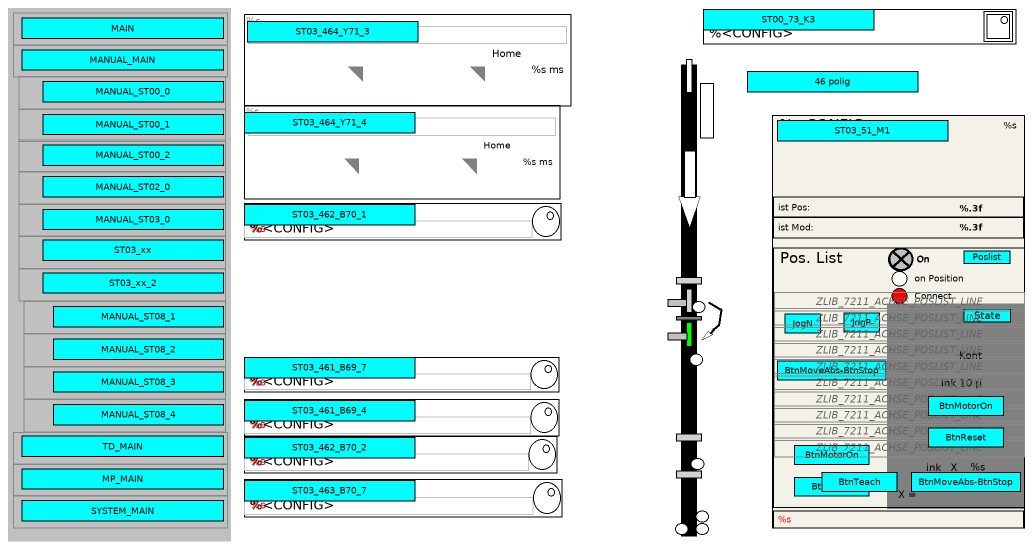
embedded screen at (3,115)-(226,648): M0000_Manual
embedded screen at (239,121)-(566,213): ZLIB_VALVE_1_SENSORS
embedded screen at (239,212)-(555,306): ZLIB_VALVE_1_SENSORS
embedded screen at (239,543)-(552,580): VDIGIN
embedded screen at (239,310)-(556,347): VDIGIN
embedded screen at (239,506)-(554,543): VDIGIN
embedded screen at (239,586)-(557,624): VDIGIN
embedded screen at (239,464)-(554,499): VDIGIN
embedded screen at (767,222)-(1021,635): ZLIB_7211_Achse
embedded screen at (646,161)-(716,643): ZUFUEHRUNG_46POL
rectangle at (742,178)-(913,199): text "46 polig"; invisible if TRUE
rectangle at (239,219)-(410,240): text "ST03_464_Y71_4"; invisible if TRUE
rectangle at (242,128)-(413,149): text "ST03_464_Y71_3"; invisible if TRUE
rectangle at (239,311)-(410,332): text "ST03_462_B70_1"; invisible if TRUE
rectangle at (239,507)-(410,528): text "ST03_461_B69_4"; invisible if TRUE
rectangle at (239,544)-(410,565): text "ST03_462_B70_2"; invisible if TRUE
rectangle at (239,587)-(410,608): text "ST03_463_B70_7"; invisible if TRUE
rectangle at (239,464)-(410,485): text "ST03_461_B69_7"; invisible if TRUE
rectangle at (772,227)-(943,248): text "ST03_51_M1"; invisible if TRUE
embedded screen at (698,116)-(1011,151): VDIGOUT_SMAL
rectangle at (698,116)-(869,137): text "ST00_73_K3"; invisible if TRUE
*)

(* Visualisation 01_ManualMode/ST03/MANUAL_ST03_9_2
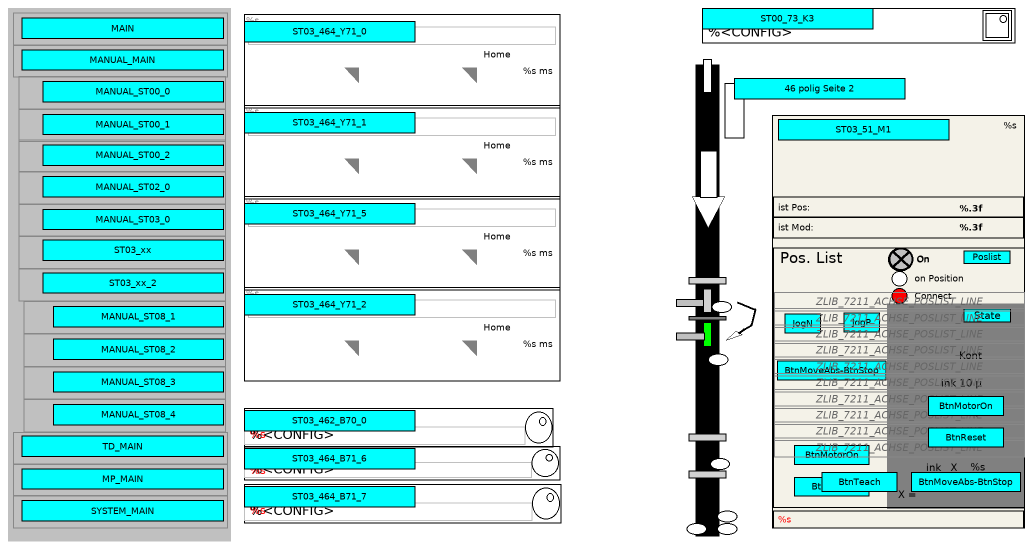
embedded screen at (3,115)-(226,648): M0000_Manual
embedded screen at (767,222)-(1021,635): ZLIB_7211_Achse
embedded screen at (646,161)-(750,643): ZUFUEHRUNG_46POL
rectangle at (729,185)-(900,206): text "46 polig Seite 2"; invisible if TRUE
embedded screen at (239,553)-(555,587): VDIGIN
embedded screen at (239,121)-(555,215): ZLIB_VALVE_1_SENSORS
rectangle at (239,128)-(410,149): text "ST03_464_Y71_0"; invisible if TRUE
rectangle at (239,555)-(410,576): text "ST03_464_B71_6"; invisible if TRUE
embedded screen at (239,212)-(555,306): ZLIB_VALVE_1_SENSORS
rectangle at (239,219)-(410,240): text "ST03_464_Y71_1"; invisible if TRUE
embedded screen at (239,394)-(555,488): ZLIB_VALVE_1_SENSORS
rectangle at (239,401)-(410,422): text "ST03_464_Y71_2"; invisible if TRUE
embedded screen at (239,303)-(555,397): ZLIB_VALVE_1_SENSORS
rectangle at (239,310)-(410,331): text "ST03_464_Y71_5"; invisible if TRUE
embedded screen at (239,515)-(548,554): VDIGIN
rectangle at (239,517)-(410,538): text "ST03_462_B70_0"; invisible if TRUE
rectangle at (773,226)-(944,247): text "ST03_51_M1"; invisible if TRUE
embedded screen at (239,591)-(556,630): VDIGIN
rectangle at (239,593)-(410,614): text "ST03_464_B71_7"; invisible if TRUE
embedded screen at (697,115)-(1010,150): VDIGOUT_SMAL
rectangle at (697,115)-(868,136): text "ST00_73_K3"; invisible if TRUE
*)

(* Visualisation 01_ManualMode/ST08/MANUAL_ST08_1
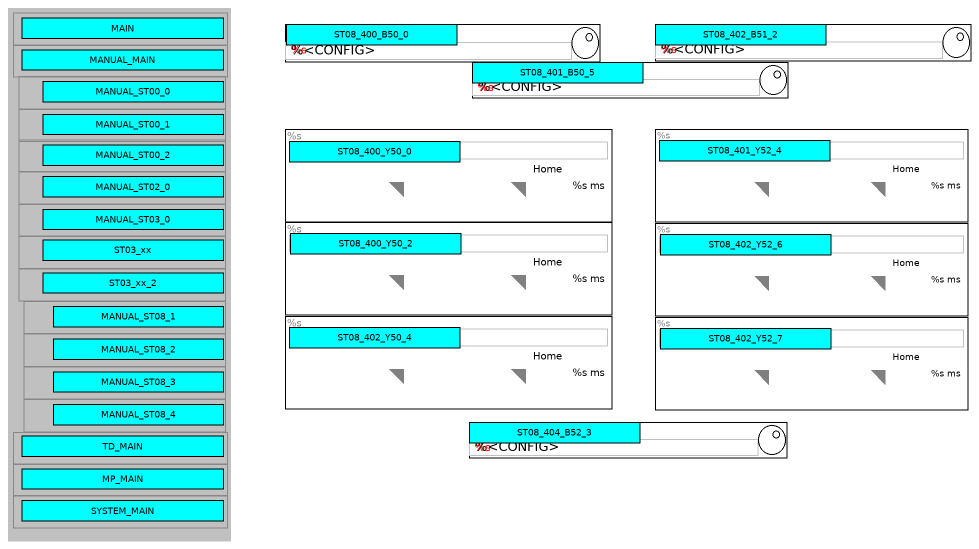
embedded screen at (3,115)-(226,648): M0000_Manual
embedded screen at (280,236)-(607,329): ZLIB_VALVE_1_SENSORS
embedded screen at (280,329)-(607,422): ZLIB_VALVE_1_SENSORS
embedded screen at (280,131)-(595,169): VDIGIN
embedded screen at (467,169)-(783,205): VDIGIN
embedded screen at (650,131)-(966,168): VDIGIN
embedded screen at (280,423)-(607,516): ZLIB_VALVE_1_SENSORS
embedded screen at (650,236)-(963,329): ZLIB_VALVE_1_SENSORS
embedded screen at (650,330)-(963,423): ZLIB_VALVE_1_SENSORS
embedded screen at (650,424)-(963,517): ZLIB_VALVE_1_SENSORS
embedded screen at (464,529)-(782,565): VDIGIN
rectangle at (281,131)-(452,152): text "ST08_400_B50_0"; invisible if TRUE
rectangle at (467,169)-(638,190): text "ST08_401_B50_5"; invisible if TRUE
rectangle at (650,131)-(821,152): text "ST08_402_B51_2"; invisible if TRUE
rectangle at (284,248)-(455,269): text "ST08_400_Y50_0"; invisible if TRUE
rectangle at (285,340)-(456,361): text "ST08_400_Y50_2"; invisible if TRUE
rectangle at (654,247)-(825,268): text "ST08_401_Y52_4"; invisible if TRUE
rectangle at (655,341)-(826,362): text "ST08_402_Y52_6"; invisible if TRUE
rectangle at (655,435)-(826,456): text "ST08_402_Y52_7"; invisible if TRUE
rectangle at (284,434)-(455,455): text "ST08_402_Y50_4"; invisible if TRUE
rectangle at (464,529)-(635,550): text "ST08_404_B52_3"; invisible if TRUE
*)

(* Visualisation 01_ManualMode/ST08/MANUAL_ST08_2
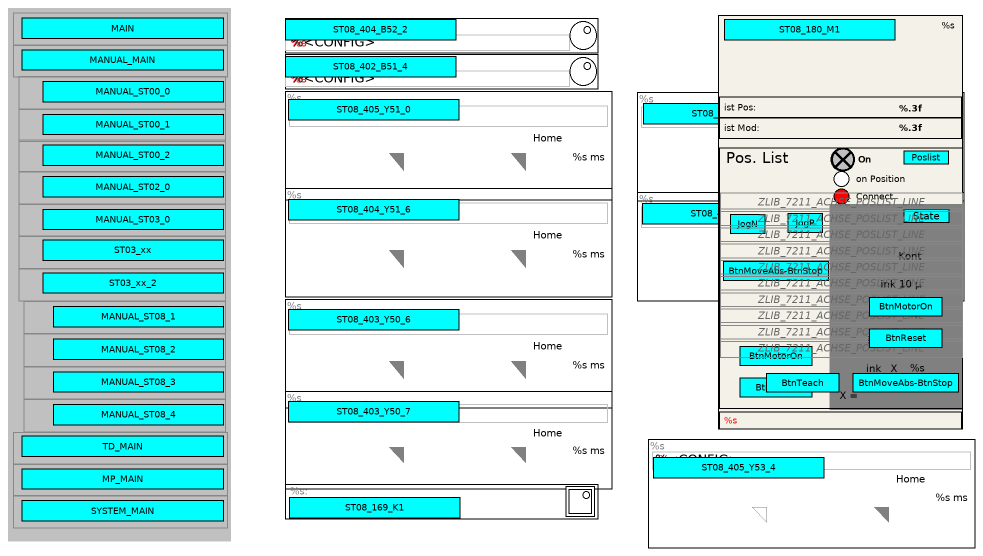
embedded screen at (3,115)-(226,648): M0000_Manual
embedded screen at (280,125)-(593,160): VDIGIN
embedded screen at (280,198)-(607,307): ZLIB_VALVE_1_SENSORS
embedded screen at (280,295)-(607,404): ZLIB_VALVE_1_SENSORS
embedded screen at (643,546)-(970,655): ZLIB_VALVE_2_SENSORS
embedded screen at (280,406)-(607,515): ZLIB_VALVE_1_SENSORS
embedded screen at (280,498)-(607,596): ZLIB_VALVE_1_SENSORS
embedded screen at (280,161)-(593,196): VDIGIN
embedded screen at (632,199)-(959,308): ZLIB_VALVE_1_SENSORS
rectangle at (638,210)-(809,231): text "ST08_404_Y53_0"; invisible if TRUE
embedded screen at (632,299)-(959,408): ZLIB_VALVE_1_SENSORS
rectangle at (637,310)-(808,331): text "ST08_404_Y53_2"; invisible if TRUE
embedded screen at (713,122)-(959,536): ZLIB_7211_Achse
embedded screen at (280,591)-(593,626): VDIGOUT_SMAL
rectangle at (280,126)-(451,147): text "ST08_404_B52_2"; invisible if TRUE
rectangle at (280,163)-(451,184): text "ST08_402_B51_4"; invisible if TRUE
rectangle at (283,206)-(454,227): text "ST08_405_Y51_0"; invisible if TRUE
rectangle at (283,306)-(454,327): text "ST08_404_Y51_6"; invisible if TRUE
rectangle at (283,416)-(454,437): text "ST08_403_Y50_6"; invisible if TRUE
rectangle at (283,508)-(454,529): text "ST08_403_Y50_7"; invisible if TRUE
rectangle at (284,604)-(455,625): text "ST08_169_K1"; invisible if TRUE
rectangle at (648,564)-(819,585): text "ST08_405_Y53_4"; invisible if TRUE
rectangle at (719,126)-(890,147): text "ST08_180_M1"; invisible if TRUE
*)

(* Visualisation 01_ManualMode/ST08/MANUAL_ST08_3
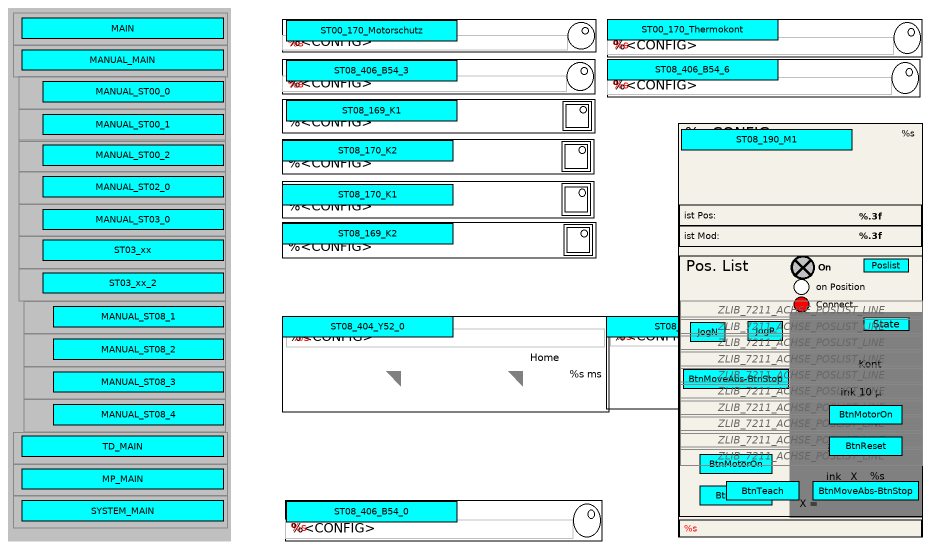
embedded screen at (3,115)-(226,648): M0000_Manual
embedded screen at (277,206)-(590,240): VDIGOUT_SMAL
embedded screen at (277,329)-(591,365): VDIGOUT_SMAL
embedded screen at (277,288)-(589,325): VDIGOUT_SMAL
embedded screen at (277,246)-(589,281): VDIGOUT_SMAL
embedded screen at (602,126)-(917,164): VDIGIN
embedded screen at (277,126)-(591,159): VDIGIN
embedded screen at (280,607)-(597,648): VDIGIN
embedded screen at (277,166)-(590,201): VDIGIN
embedded screen at (601,423)-(914,516): ZLIB_VALVE_1_SENSORS
embedded screen at (277,423)-(604,519): ZLIB_VALVE_1_SENSORS
rectangle at (601,423)-(772,444): text "ST08_406_Y52_3"; invisible if TRUE
rectangle at (277,423)-(448,444): text "ST08_404_Y52_0"; invisible if TRUE
rectangle at (281,207)-(452,228): text "ST08_169_K1"; invisible if TRUE
rectangle at (277,330)-(448,351): text "ST08_169_K2"; invisible if TRUE
rectangle at (277,291)-(448,312): text "ST08_170_K1"; invisible if TRUE
rectangle at (277,247)-(448,268): text "ST08_170_K2"; invisible if TRUE
rectangle at (281,127)-(452,148): text "ST00_170_Motorschutz"; invisible if TRUE
rectangle at (602,126)-(773,147): text "ST00_170_Thermokont"; invisible if TRUE
rectangle at (281,608)-(452,629): text "ST08_406_B54_0"; invisible if TRUE
rectangle at (281,167)-(452,188): text "ST08_406_B54_3"; invisible if TRUE
embedded screen at (602,166)-(915,204): VDIGIN
rectangle at (602,166)-(773,187): text "ST08_406_B54_6"; invisible if TRUE
embedded screen at (673,230)-(919,644): ZLIB_7211_Achse
rectangle at (676,236)-(847,257): text "ST08_190_M1"; invisible if TRUE
*)

(* Visualisation 01_ManualMode/ST08/MANUAL_ST08_4
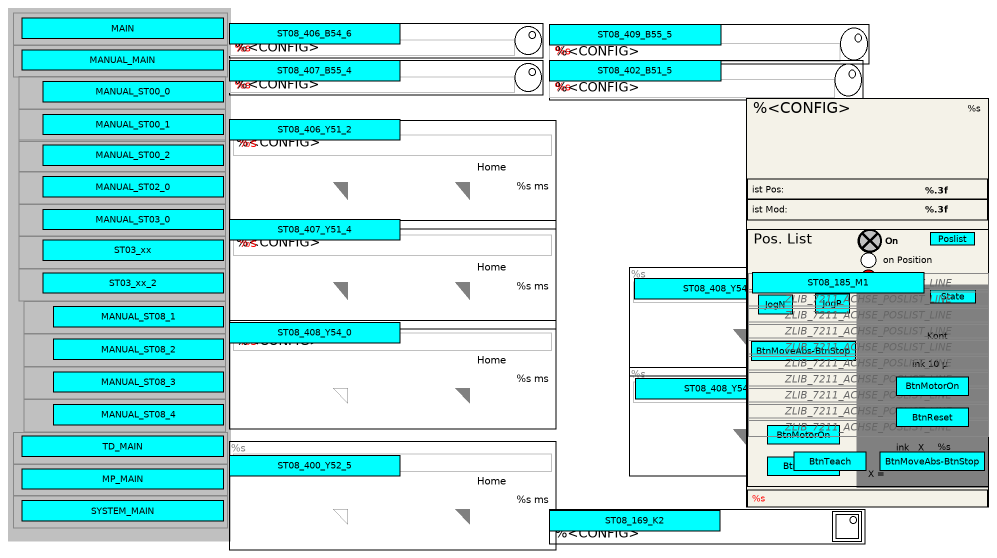
embedded screen at (3,115)-(226,648): M0000_Manual
embedded screen at (224,427)-(551,536): ZLIB_VALVE_2_SENSORS
embedded screen at (224,130)-(538,165): VDIGIN
embedded screen at (224,227)-(551,336): ZLIB_VALVE_1_SENSORS
embedded screen at (224,327)-(551,436): ZLIB_VALVE_1_SENSORS
embedded screen at (544,131)-(864,171): VDIGIN
embedded screen at (224,548)-(551,657): ZLIB_VALVE_2_SENSORS
embedded screen at (544,167)-(858,207): VDIGIN
embedded screen at (624,374)-(951,483): ZLIB_VALVE_1_SENSORS
rectangle at (629,385)-(801,406): text "ST08_408_Y54_2"; invisible if TRUE
embedded screen at (624,474)-(951,583): ZLIB_VALVE_1_SENSORS
rectangle at (630,485)-(802,506): text "ST08_408_Y54_4"; invisible if TRUE
embedded screen at (741,205)-(985,614): ZLIB_7211_Achse
embedded screen at (224,167)-(538,202): VDIGIN
embedded screen at (544,616)-(860,651): VDIGOUT_SMAL
rectangle at (224,562)-(395,583): text "ST08_400_Y52_5"; invisible if TRUE
rectangle at (544,617)-(715,638): text "ST08_169_K2"; invisible if TRUE
rectangle at (224,429)-(395,450): text "ST08_408_Y54_0"; invisible if TRUE
rectangle at (224,326)-(395,347): text "ST08_407_Y51_4"; invisible if TRUE
rectangle at (224,226)-(395,247): text "ST08_406_Y51_2"; invisible if TRUE
rectangle at (224,130)-(395,151): text "ST08_406_B54_6"; invisible if TRUE
rectangle at (224,167)-(395,188): text "ST08_407_B55_4"; invisible if TRUE
rectangle at (544,131)-(716,152): text "ST08_409_B55_5"; invisible if TRUE
rectangle at (544,167)-(716,188): text "ST08_402_B51_5"; invisible if TRUE
rectangle at (747,379)-(919,400): text "ST08_185_M1"; invisible if TRUE
*)

(* Visualisation 00_Main/MASTER_MAIN
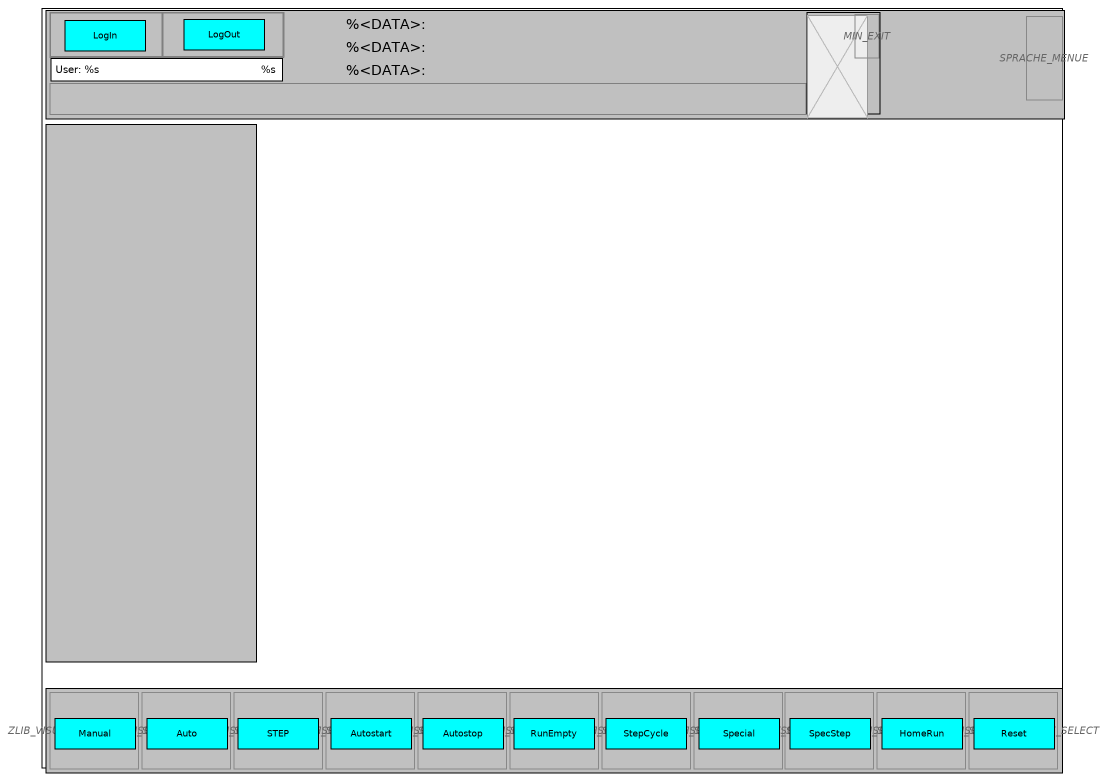
embedded screen at (8,684)-(97,761): ZLIB_VISUBUTTON_MODE_SELECT
embedded screen at (100,684)-(189,761): ZLIB_VISUBUTTON_MODE_SELECT
embedded screen at (192,684)-(281,761): ZLIB_VISUBUTTON_MODE_SELECT
embedded screen at (284,684)-(373,761): ZLIB_VISUBUTTON_MODE_SELECT
embedded screen at (376,684)-(465,761): ZLIB_VISUBUTTON_MODE_SELECT
embedded screen at (468,684)-(557,761): ZLIB_VISUBUTTON_MODE_SELECT
embedded screen at (560,684)-(649,761): ZLIB_VISUBUTTON_MODE_SELECT
embedded screen at (652,684)-(741,761): ZLIB_VISUBUTTON_MODE_SELECT
embedded screen at (835,684)-(924,761): ZLIB_VISUBUTTON_MODE_SELECT
embedded screen at (927,684)-(1016,761): ZLIB_VISUBUTTON_MODE_SELECT
rectangle at (247,29)-(386,49): text "%<DATA>:"; shows 'ArtNo'
rectangle at (247,6)-(386,26): text "%<DATA>:"; shows 'TypeName'
rectangle at (247,52)-(386,72): text "%<DATA>:"; shows 'TypeDescription'
rectangle at (9,50)-(241,73): text "User: %s"; shows UserLoginHandler.CurrentUser.UserName
embedded screen at (8,4)-(121,49): ZLIB_VISUBUTTON_S18
embedded screen at (120,4)-(242,49): ZLIB_VISUBUTTON_S18
embedded screen at (8,75)-(764,106): ZLIB_ShowMessageButton
embedded screen at (743,684)-(832,761): ZLIB_VISUBUTTON_MODE_SELECT
rectangle at (13,710)-(94,741): text "Manual"; invisible if TRUE
rectangle at (105,710)-(186,741): text "Auto"; invisible if TRUE
rectangle at (196,710)-(277,741): text "STEP"; invisible if TRUE
rectangle at (289,710)-(370,741): text "Autostart"; invisible if TRUE
rectangle at (381,710)-(462,741): text "Autostop"; invisible if TRUE
rectangle at (472,710)-(553,741): text "RunEmpty"; invisible if TRUE
rectangle at (564,710)-(645,741): text "StepCycle"; invisible if TRUE
rectangle at (657,710)-(738,741): text "Special"; invisible if TRUE
rectangle at (748,710)-(829,741): text "SpecStep"; invisible if TRUE
rectangle at (840,710)-(921,741): text "HomeRun"; invisible if TRUE
rectangle at (932,710)-(1013,741): text "Reset"; invisible if TRUE
rectangle at (142,11)-(223,42): text "LogOut"; invisible if TRUE
rectangle at (23,12)-(104,43): text "LogIn"; invisible if TRUE
rectangle at (157,52)-(239,71): text "%s"; shows UserLoginHandler.s_AutoLoggedOut
group at (765,4)-(1021,110)
  bitmap at (3,3)-(213,106): c:\twincat\plc\VisuBmp\ept_logo.jpg
  embedded screen at (168,2)-(253,46): MIN_EXIT
  embedded screen at (765,4)-(891,88): SPRACHE_MENUE
5 more shapes without text or variables
6 elements of other kinds (tables, trends, ...) not read
*)

(* Visualisation zLibrary/ept/MIN_EXIT
2 elements of other kinds (tables, trends, ...) not read
*)

(* Visualisation 03_MachPara/MP_DATE
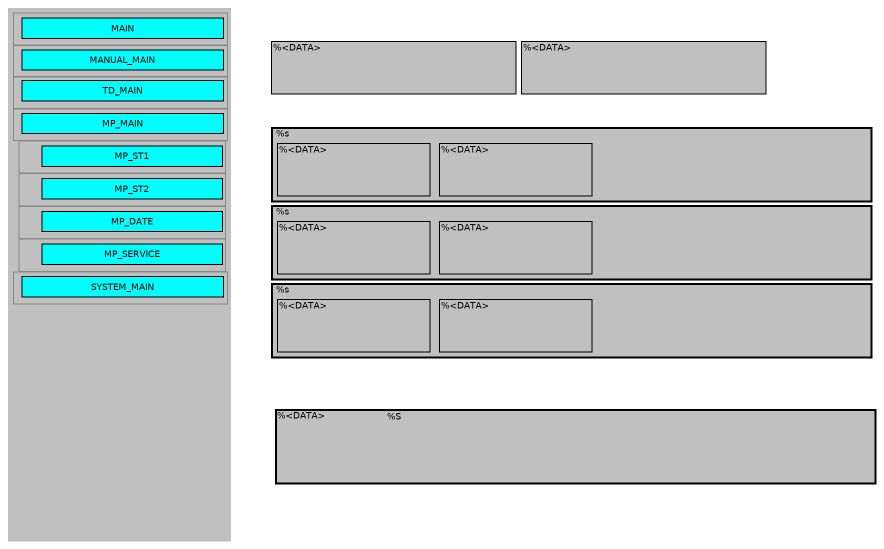
rectangle at (266,390)-(867,465): text "%s"; shows .MP.ShiftData.Shift[3].ShiftName; alarm colour if .MP.ShiftData.Shift[3].ShiftActive
rectangle at (266,312)-(867,387): text "%s"; shows .MP.ShiftData.Shift[2].ShiftName; alarm colour if .MP.ShiftData.Shift[2].ShiftActive
rectangle at (266,234)-(867,309): text "%s"; shows .MP.ShiftData.Shift[1].ShiftName; alarm colour if .MP.ShiftData.Shift[1].ShiftActive
rectangle at (516,148)-(761,201): text "%<DATA>"; shows 'Uhrzeit'
rectangle at (266,148)-(511,201): text "%<DATA>"; shows 'Datum'
embedded screen at (3,115)-(226,648): M0002_Machpara
rectangle at (272,250)-(425,303): text "%<DATA>"; shows 'Uhrzeit Start'
rectangle at (434,250)-(587,303): text "%<DATA>"; shows 'Uhrzeit Ende'
rectangle at (272,328)-(425,381): text "%<DATA>"; shows 'Uhrzeit Start'
rectangle at (434,328)-(587,381): text "%<DATA>"; shows 'Uhrzeit Ende'
rectangle at (272,406)-(425,459): text "%<DATA>"; shows 'Uhrzeit Start'
rectangle at (434,406)-(587,459): text "%<DATA>"; shows 'Uhrzeit Ende'
rectangle at (270,516)-(871,591): text "%<DATA>"; shows 'Aktuelle Schicht'; alarm colour if .MP.ShiftData.Activeshift.ShiftActive
rectangle at (380,515)-(511,532): text "%S"; shows .MP.ShiftData.Activeshift.ShiftName
35 elements of other kinds (tables, trends, ...) not read
*)

(* Visualisation 03_MachPara/MP_SERVICE
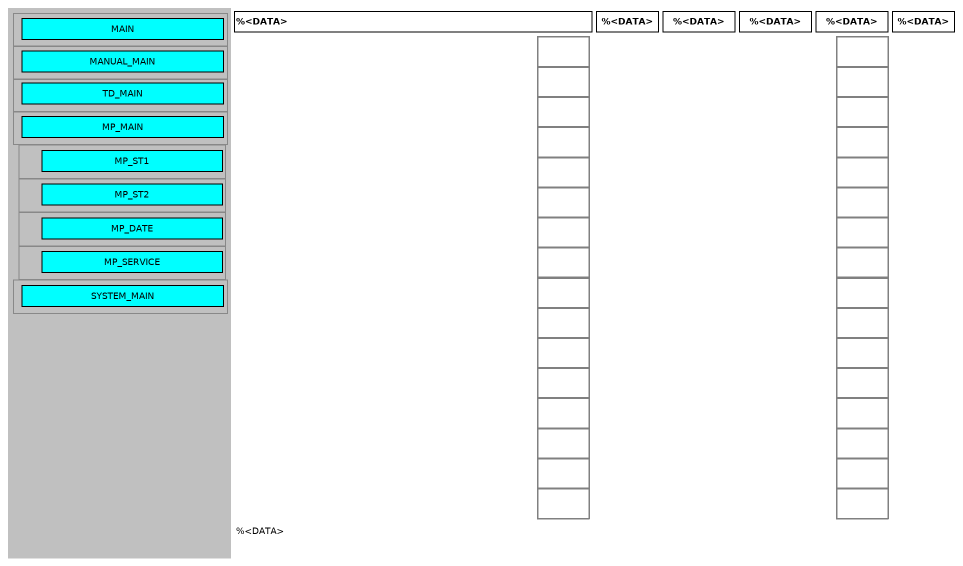
embedded screen at (3,115)-(226,665): M0002_Machpara
embedded screen at (229,118)-(1011,651): ZLIB_SERVICELIST
*)

(* Visualisation 03_MachPara/MP_ST1
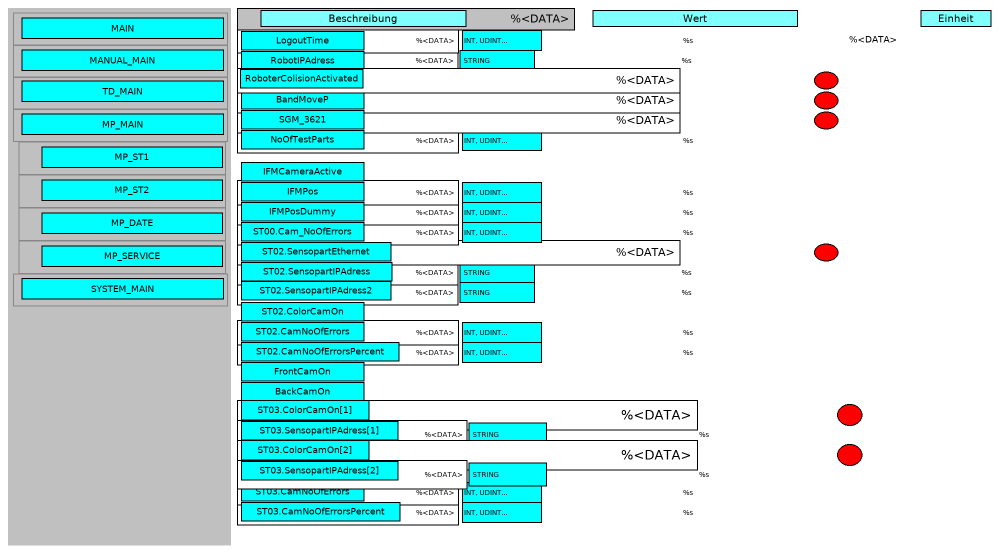
embedded screen at (3,115)-(226,652): M0002_Machpara
rectangle at (842,136)-(960,157): text "%<DATA>"; shows '0_deaktiv'
embedded screen at (232,607)-(833,632): Data_DEZIMAL
embedded screen at (232,587)-(833,612): Data_DEZIMAL
embedded screen at (232,447)-(833,472): Data_DEZIMAL
embedded screen at (232,427)-(833,452): Data_DEZIMAL
embedded screen at (232,387)-(833,412): Data_STRING
embedded screen at (232,367)-(833,392): Data_STRING
embedded screen at (232,347)-(833,372): Data_BOOL
embedded screen at (232,327)-(833,352): Data_DEZIMAL
embedded screen at (232,307)-(833,332): Data_DEZIMAL
embedded screen at (232,287)-(833,312): Data_DEZIMAL
embedded screen at (232,235)-(833,260): Data_DEZIMAL
embedded screen at (232,215)-(833,240): Data_BOOL
embedded screen at (232,195)-(833,220): Data_BOOL
embedded screen at (232,155)-(833,180): Data_STRING
embedded screen at (232,135)-(833,160): Data_DEZIMAL
rectangle at (236,158)-(359,177): text "RobotIPAdress"; invisible if TRUE
rectangle at (236,197)-(359,216): text "BandMoveP"; invisible if TRUE
rectangle at (236,217)-(359,236): text "SGM_3621"; invisible if TRUE
rectangle at (236,369)-(387,388): text "ST02.SensopartIPAdress"; invisible if TRUE
rectangle at (236,349)-(386,368): text "ST02.SensopartEthernet"; invisible if TRUE
rectangle at (236,269)-(359,288): text "IFMCameraActive"; invisible if TRUE
rectangle at (236,309)-(359,328): text "IFMPosDummy"; invisible if TRUE
rectangle at (236,388)-(386,407): text "ST02.SensopartIPAdress2"; invisible if TRUE
rectangle at (236,449)-(394,468): text "ST02.CamNoOfErrorsPercent"; invisible if TRUE
rectangle at (236,469)-(359,488): text "FrontCamOn"; invisible if TRUE
rectangle at (236,609)-(395,628): text "ST03.CamNoOfErrorsPercent"; invisible if TRUE
rectangle at (236,237)-(359,256): text "NoOfTestParts"; invisible if TRUE
rectangle at (236,329)-(359,348): text "ST00.Cam_NoOfErrors"; invisible if TRUE
rectangle at (236,429)-(359,448): text "ST02.CamNoOfErrors"; invisible if TRUE
rectangle at (236,489)-(359,508): text "BackCamOn"; shows 'BackCamOn'; invisible if TRUE
rectangle at (236,589)-(359,608): text "ST03.CamNoOfErrors"; invisible if TRUE
rectangle at (236,289)-(359,308): text "IFMPos"; invisible if TRUE
rectangle at (236,138)-(359,157): text "LogoutTime"; invisible if TRUE
rectangle at (236,409)-(359,428): text "ST02.ColorCamOn"; invisible if TRUE
embedded screen at (232,175)-(833,200): Data_BOOL
rectangle at (235,176)-(358,195): text "RoboterColisionActivated"; shows 'BackCamOn'; invisible if TRUE
embedded screen at (232,115)-(986,137): DATA_HEADER_BEER
embedded screen at (232,507)-(857,537): Data_BOOL
embedded screen at (232,527)-(857,556): Data_STRING
rectangle at (236,528)-(393,547): text "ST03.SensopartIPAdress[1]"; invisible if TRUE
rectangle at (236,507)-(364,527): text "ST03.ColorCamOn[1]"; invisible if TRUE
embedded screen at (232,547)-(857,577): Data_BOOL
embedded screen at (232,567)-(857,596): Data_STRING
rectangle at (236,568)-(393,587): text "ST03.SensopartIPAdress[2]"; invisible if TRUE
rectangle at (236,547)-(364,567): text "ST03.ColorCamOn[2]"; invisible if TRUE
4 elements of other kinds (tables, trends, ...) not read
*)

(* Visualisation 03_MachPara/MP_ST2
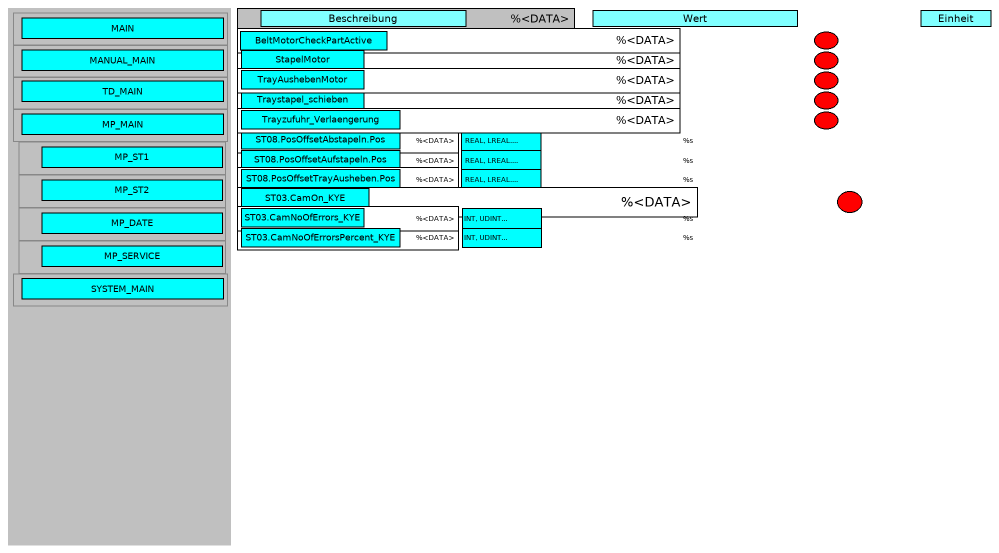
embedded screen at (3,115)-(226,652): M0002_Machpara
embedded screen at (232,115)-(986,137): DATA_HEADER_BEER
embedded screen at (232,255)-(833,280): Data_DEZIMAL_REAL
embedded screen at (232,235)-(833,260): Data_DEZIMAL_REAL
embedded screen at (232,195)-(833,220): Data_BOOL
embedded screen at (232,155)-(833,180): Data_BOOL
embedded screen at (232,135)-(833,160): Data_BOOL
rectangle at (236,197)-(359,216): text "Traystapel_schieben"; invisible if TRUE
rectangle at (236,157)-(359,176): text "StapelMotor"; invisible if TRUE
rectangle at (236,237)-(395,256): text "ST08.PosOffsetAbstapeln.Pos"; invisible if TRUE
rectangle at (236,257)-(395,276): text "ST08.PosOffsetAufstapeln.Pos"; invisible if TRUE
rectangle at (235,138)-(382,157): text "BeltMotorCheckPartActive"; invisible if TRUE
embedded screen at (232,175)-(833,200): Data_BOOL
rectangle at (236,177)-(359,196): text "TrayAushebenMotor"; invisible if TRUE
embedded screen at (232,274)-(833,299): Data_DEZIMAL_REAL
rectangle at (236,276)-(395,295): text "ST08.PosOffsetTrayAusheben.Pos"; invisible if TRUE
embedded screen at (232,215)-(833,240): Data_BOOL
rectangle at (236,217)-(395,236): text "Trayzufuhr_Verlaengerung"; invisible if TRUE
embedded screen at (232,294)-(857,324): Data_BOOL
rectangle at (236,295)-(364,315): text "ST03.CamOn_KYE"; invisible if TRUE
embedded screen at (232,332)-(833,357): Data_DEZIMAL
embedded screen at (232,313)-(833,338): Data_DEZIMAL
rectangle at (236,335)-(395,354): text "ST03.CamNoOfErrorsPercent_KYE"; invisible if TRUE
rectangle at (236,315)-(359,334): text "ST03.CamNoOfErrors_KYE"; invisible if TRUE
*)

(* Visualisation zLibrary/X_MachSpec/PARTRESULT
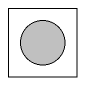
ellipse at (12,12)-(57,57): invisible if ($PartResult$ MOD 10) = 0; alarm colour if ($PartResult$ MOD 10) <> 1
ellipse at (12,12)-(57,57): invisible if ($PartResult$ MOD 10) <> 4
ellipse at (12,12)-(57,57): invisible if ($PartResult$ MOD 10) <> 5
ellipse at (12,12)-(57,57): invisible if ($PartResult$ MOD 10) <> 0
1 more shapes without text or variables
*)

(* Visualisation zLibrary/ept/Pruefteile/PRUEFTEILEN_CZ
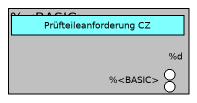
rectangle at (0,0)-(181,86): text "%<BASIC>"; shows 'auto_Prüfteileanforderung'
rectangle at (156,37)-(179,59): text "%d"; shows ST03_Main.CTR; invisible if gTakeTestParts=FALSE AND gTakeTestPartsAuto=FALSE; alarm colour if gTakeTestParts OR gTakeTestPartsAuto
rectangle at (18,61)-(153,82): text "%<BASIC>"; shows 'Rutsche belegt'; invisible if .TD.TestpartBilister
ellipse at (156,61)-(167,72): invisible if .TD.TestpartBilister; alarm colour if ST03_8_75_B13_5.BitInToCheck
ellipse at (156,73)-(167,84): invisible if .TD.TestpartBilister; alarm colour if ST03_8_75_B13_6.BitInToCheck
rectangle at (3,7)-(176,27): text "Prüfteileanforderung CZ"; invisible if TRUE
1 elements of other kinds (tables, trends, ...) not read
*)

(* Visualisation zLibrary/ept/Pruefteile/PRUEFTEILEN_DE
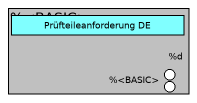
rectangle at (0,0)-(181,86): text "%<BASIC>"; shows 'Prüfteileanforderung'
rectangle at (156,37)-(179,59): text "%d"; shows ST03_Main.CTR; invisible if gTakeTestParts=FALSE AND gTakeTestPartsAuto=FALSE; alarm colour if gTakeTestParts OR gTakeTestPartsAuto
rectangle at (19,61)-(153,82): text "%<BASIC>"; shows 'Rutsche belegt'; invisible if .TD.TestpartBilister
ellipse at (156,61)-(167,72): invisible if .TD.TestpartBilister; alarm colour if ST03_8_75_B13_5.BitInToCheck
ellipse at (156,73)-(167,84): invisible if .TD.TestpartBilister; alarm colour if ST03_8_75_B13_6.BitInToCheck
rectangle at (3,7)-(176,27): text "Prüfteileanforderung DE"; invisible if TRUE
1 elements of other kinds (tables, trends, ...) not read
*)

(* Visualisation zLibrary/ept/Pruefteile/PRUEFTEILENTNAHME
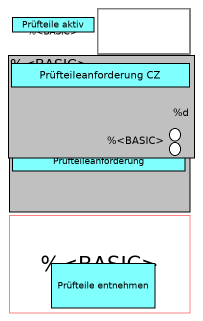
embedded screen at (89,5)-(182,51): ZLIB_VISUBUTTON_S24
rectangle at (1,8)-(88,49): text "%<BASIC>"; shows 'Prüfteile aktiv'; invisible if NOT gTakeTestParts AND NOT gTakeTestPartsAuto; alarm colour if gTakeTestParts OR gTakeTestPartsAuto
rectangle at (1,212)-(182,310): text "%<BASIC>"; shows 'Prüfteile entnehmen'; invisible if NOT ST03_Main.TestPartsRemove; taps gTakeTestPartsFinished
rectangle at (43,260)-(147,305): text "Prüfteile entnehmen"; invisible if TRUE
rectangle at (4,14)-(86,29): text "Prüfteile aktiv"; invisible if TRUE
rectangle at (1,141)-(182,209): text "%<BASIC>"; shows 'Teile seit letzten Test'
rectangle at (4,148)-(177,168): text "Prüfteileanforderung"; invisible if TRUE
embedded screen at (0,52)-(187,155): PRUEFTEILEN_CZ
2 elements of other kinds (tables, trends, ...) not read
*)

(* Visualisation zLibrary/X_MachSpec/RoundTable/ROUNDTABLE
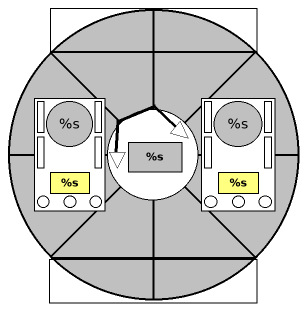
polyline at (147,3)-(147,291): invisible if (ST02_DT_62_B81.ValveSensor OR ST02_DT_62_B91.ValveSensor)
polyline at (2,147)-(292,147): invisible if (ST02_DT_62_B81.ValveSensor OR ST02_DT_62_B91.ValveSensor)
polyline at (44,44)-(249,249): invisible if NOT (ST02_DT_62_B81.ValveSensor OR ST02_DT_62_B91.ValveSensor)
polyline at (44,44)-(249,249): invisible if NOT (ST02_DT_62_B81.ValveSensor OR ST02_DT_62_B91.ValveSensor)
embedded screen at (195,90)-(269,203): RoundTableNest
embedded screen at (28,90)-(99,203): ROUNDTABLENEST
polygon at (103,144)-(119,160): alarm colour if ST02_62_Y6.MoveWork
rounded rectangle at (122,134)-(176,164): text "%s"; shows MachineStates.CycleTimeHelp
polygon at (164,113)-(182,130): alarm colour if ST02_62_Y6.MoveInit
7 more shapes without text or variables
*)

(* Visualisation zLibrary/X_MachSpec/RoundTable/ROUNDTABLE_1
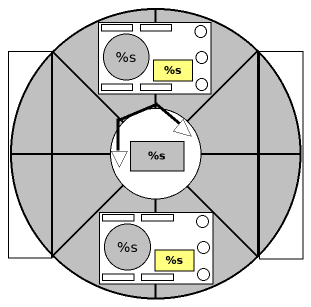
polyline at (147,3)-(147,291): invisible if (ST02_DT_62_B81.ValveSensor OR ST02_DT_62_B91.ValveSensor)
polyline at (2,147)-(292,147): invisible if (ST02_DT_62_B81.ValveSensor OR ST02_DT_62_B91.ValveSensor)
polyline at (44,44)-(249,249): invisible if NOT (ST02_DT_62_B81.ValveSensor OR ST02_DT_62_B91.ValveSensor)
polyline at (44,44)-(249,249): invisible if NOT (ST02_DT_62_B81.ValveSensor OR ST02_DT_62_B91.ValveSensor)
embedded screen at (90,14)-(203,87): RoundTableNest_1
embedded screen at (91,204)-(205,277): ROUNDTABLENEST_1
polygon at (103,144)-(119,160): alarm colour if ST02_62_Y6.MoveWork
rounded rectangle at (122,134)-(176,164): text "%s"; shows MachineStates.CycleTimeHelp
polygon at (165,112)-(183,129): alarm colour if ST02_62_Y6.MoveInit
7 more shapes without text or variables
*)

(* Visualisation zLibrary/X_MachSpec/RoundTable/ROUNDTABLENEST
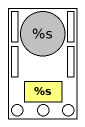
ellipse at (12,3)-(57,48): text "%s"; shows $NestNo$; invisible if NOT MP.ST02.TableData[$NestNo$].ProcessData.Part; alarm colour if MP.ST02.TableData[$NestNo$].ProcessData.Result >11; toggles MP.ST02.TableData[$NestNo$].ProcessData.Part
ellipse at (12,3)-(57,48): text "%s"; shows $NestNo$; invisible if MP.ST02.TableData[$NestNo$].ProcessData.Part; toggles MP.ST02.TableData[$NestNo$].ProcessData.Part
rectangle at (16,73)-(54,94): text "%s"; shows MP.ST02.TableData[$NestNo$].ProcessData.Result; editable
rectangle at (3,38)-(10,69): invisible if NOT MP.ST02.TableData[$NestNo$].ProcessData.Part OR MP.ST02.TableData[$NestNo$].ProcessData.Result >=19; alarm colour if MP.ST02.TableData[$NestNo$].ProcessData.Result >=1
rectangle at (3,3)-(10,34): invisible if NOT MP.ST02.TableData[$NestNo$].ProcessData.Part OR MP.ST02.TableData[$NestNo$].ProcessData.Result >=19; alarm colour if MP.ST02.TableData[$NestNo$].ProcessData.Result >=1
rectangle at (59,38)-(66,69): invisible if NOT MP.ST02.TableData[$NestNo$].ProcessData.Part OR MP.ST02.TableData[$NestNo$].ProcessData.Result >=19; alarm colour if MP.ST02.TableData[$NestNo$].ProcessData.Result >=11
rectangle at (59,3)-(66,34): invisible if NOT MP.ST02.TableData[$NestNo$].ProcessData.Part OR MP.ST02.TableData[$NestNo$].ProcessData.Result >=19; alarm colour if MP.ST02.TableData[$NestNo$].ProcessData.Result >=11
ellipse at (3,96)-(15,108): invisible if MP.ST02.TableData[$NestNo$].ProcessData.Nest_Nr = 0; alarm colour if ST02_Schwenkarm[MP.ST02.TableData[$NestNo$].ProcessData.Nest_Nr].ST02_90_0_sens
ellipse at (29,96)-(41,108): invisible if MP.ST02.TableData[$NestNo$].ProcessData.Nest_Nr = 0; alarm colour if ST02_Schwenkarm[MP.ST02.TableData[$NestNo$].ProcessData.Nest_Nr].ST02_90_sens
ellipse at (54,96)-(66,108): invisible if MP.ST02.TableData[$NestNo$].ProcessData.Nest_Nr = 0; alarm colour if ST02_Schwenkarm[MP.ST02.TableData[$NestNo$].ProcessData.Nest_Nr].ST02_90_180_sens
1 more shapes without text or variables
1 elements of other kinds (tables, trends, ...) not read
*)

(* Visualisation zLibrary/X_MachSpec/RoundTable/ROUNDTABLENEST_1
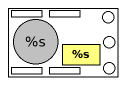
ellipse at (5,12)-(50,57): text "%s"; shows $NestNo$; invisible if NOT MP.ST02.TableData[$NestNo$].ProcessData.Part; alarm colour if MP.ST02.TableData[$NestNo$].ProcessData.Result >=99; toggles MP.ST02.TableData[$NestNo$].ProcessData.Part
ellipse at (5,12)-(50,57): text "%s"; shows $NestNo$; invisible if MP.ST02.TableData[$NestNo$].ProcessData.Part; toggles MP.ST02.TableData[$NestNo$].ProcessData.Part
rectangle at (54,37)-(92,58): text "%s"; shows MP.ST02.TableData[$NestNo$].ProcessData.Result; editable
rectangle at (41,60)-(72,67): invisible if NOT MP.ST02.TableData[$NestNo$].ProcessData.Part OR MP.ST02.TableData[$NestNo$].ProcessData.Result >=19; alarm colour if MP.ST02.TableData[$NestNo$].ProcessData.Result >=1
rectangle at (3,60)-(34,67): invisible if NOT MP.ST02.TableData[$NestNo$].ProcessData.Part OR MP.ST02.TableData[$NestNo$].ProcessData.Result >=19; alarm colour if MP.ST02.TableData[$NestNo$].ProcessData.Result >=1
rectangle at (41,3)-(72,10): invisible if NOT MP.ST02.TableData[$NestNo$].ProcessData.Part OR MP.ST02.TableData[$NestNo$].ProcessData.Result >=19; alarm colour if MP.ST02.TableData[$NestNo$].ProcessData.Result >=11
rectangle at (3,3)-(34,10): invisible if NOT MP.ST02.TableData[$NestNo$].ProcessData.Part OR MP.ST02.TableData[$NestNo$].ProcessData.Result >=19; alarm colour if MP.ST02.TableData[$NestNo$].ProcessData.Result >=11
ellipse at (95,55)-(107,67): invisible if MP.ST02.TableData[$NestNo$].ProcessData.Nest_Nr = 0; alarm colour if ST02_Schwenkarm[MP.ST02.TableData[$NestNo$].ProcessData.Nest_Nr].ST02_90_0_sens
ellipse at (95,29)-(107,41): invisible if MP.ST02.TableData[$NestNo$].ProcessData.Nest_Nr = 0; alarm colour if ST02_Schwenkarm[MP.ST02.TableData[$NestNo$].ProcessData.Nest_Nr].ST02_90_sens
ellipse at (94,4)-(106,16): invisible if MP.ST02.TableData[$NestNo$].ProcessData.Nest_Nr = 0; alarm colour if ST02_Schwenkarm[MP.ST02.TableData[$NestNo$].ProcessData.Nest_Nr].ST02_90_180_sens
1 more shapes without text or variables
1 elements of other kinds (tables, trends, ...) not read
*)

(* Visualisation zLibrary/X_MachSpec/RoundTable/ROUNDTABLENESTNR
ellipse at (0,0)-(45,45): text "%s"; shows MP.ST02.TableData[$NestNo$].ProcessData.Nest_Nr; alarm colour if MP.ST02.DeactivatedNests[MP.ST02.TableData[$NestNo$].ProcessData.Nest_Nr]
*)

(* Visualisation zLibrary/X_MachSpec/Signs/SIGNS_ARROWDOWN
polygon at (0,72)-(48,120): alarm colour if $OnBit$
rectangle at (12,0)-(37,73): alarm colour if $OnBit$
*)

(* Visualisation zLibrary/X_MachSpec/Signs/SIGNS_ARROWLEFT
polygon at (0,0)-(48,48): alarm colour if $OnBit$
rectangle at (48,12)-(121,37): alarm colour if $OnBit$
*)

(* Visualisation zLibrary/X_MachSpec/Signs/SIGNS_ARROWRIGHT
polygon at (72,0)-(120,48): alarm colour if $OnBit$
rectangle at (0,12)-(73,37): alarm colour if $OnBit$
*)

(* Visualisation zLibrary/X_MachSpec/Signs/SIGNS_ARROWUP
polygon at (0,0)-(48,48): alarm colour if $OnBit$
rectangle at (12,48)-(37,121): alarm colour if $OnBit$
*)

(* Visualisation zLibrary/ept/Axis/SIGNS_AXIS
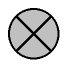
ellipse at (0,0)-(51,51): alarm colour if $Object$.on
polyline at (8,8)-(43,43): angle $Object$.sPos.lr_Mod /4
polyline at (8,8)-(43,43): angle $Object$.sPos.lr_Mod /4
*)

(* Visualisation zLibrary/ept/TippiDrucker/SIGNS_PUMP
3 elements of other kinds (tables, trends, ...) not read
*)

(* Visualisation zLibrary/ept/SPRACHE_MENUE
14 elements of other kinds (tables, trends, ...) not read
*)

(* Visualisation 04_System/SYSTEM_ERRORLIST
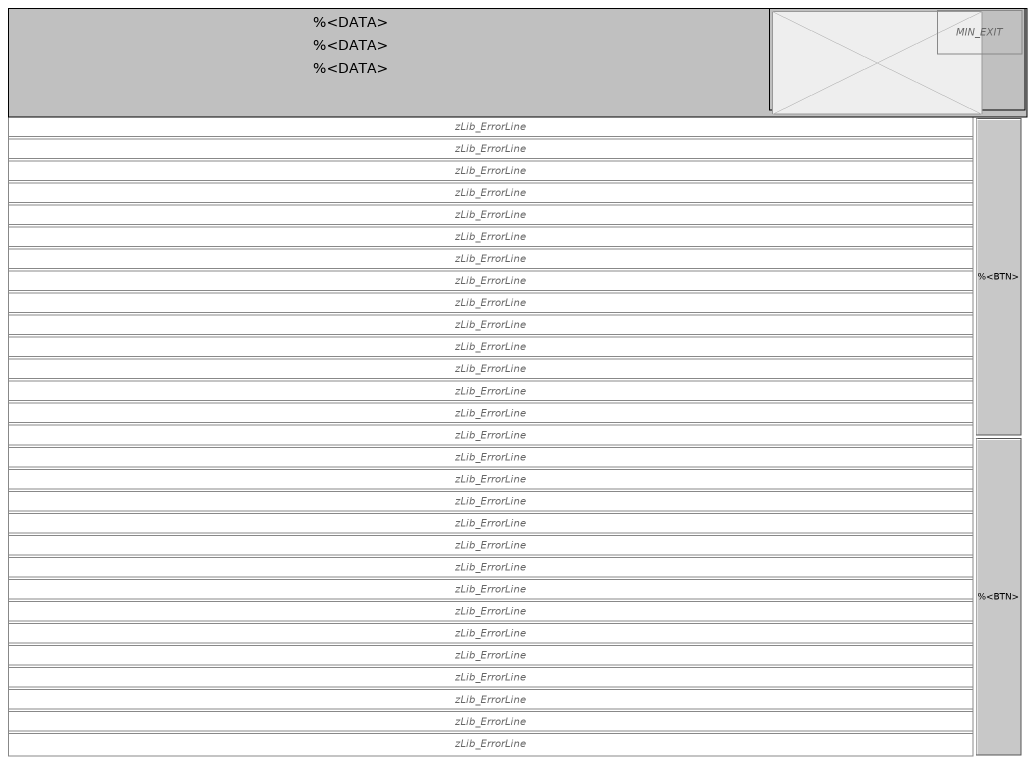
embedded screen at (4,112)-(969,754): zLib_ErrorList
button at (972,116)-(1017,433): text "%<BTN>"; shows 'up'; runs INTERN ASSIGN Visu.ErrorHistoryScroll:=(Visu.ErrorHistoryScroll - 29)
button at (972,436)-(1017,753): text "%<BTN>"; shows 'down'; runs INTERN ASSIGN Visu.ErrorHistoryScroll:=(Visu.ErrorHistoryScroll + 29)
rectangle at (0,114)-(971,765): opens ZOOMTOCALLER
rectangle at (248,50)-(387,67): shows 'TypeDescription'
bitmap at (768,9)-(978,112): c:\twincat\plc\VisuBmp\ept_logo.jpg
embedded screen at (933,8)-(1018,52): MIN_EXIT
rectangle at (247,33)-(386,53): text "%<DATA>"; shows 'ArtNo'
rectangle at (247,10)-(386,30): text "%<DATA>"; shows 'TypeName'
rectangle at (247,56)-(386,76): text "%<DATA>"; shows 'TypeDescription'
2 more shapes without text or variables
4 elements of other kinds (tables, trends, ...) not read
*)

(* Visualisation 04_System/SYSTEM_FEATURES
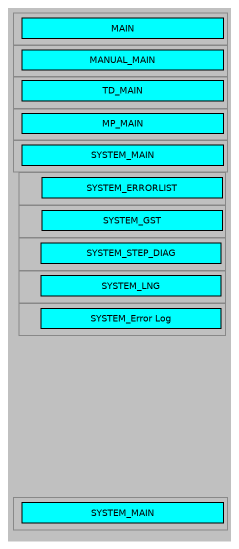
embedded screen at (3,115)-(226,648): M0003_System
*)

(* Visualisation 04_System/SYSTEM_GST
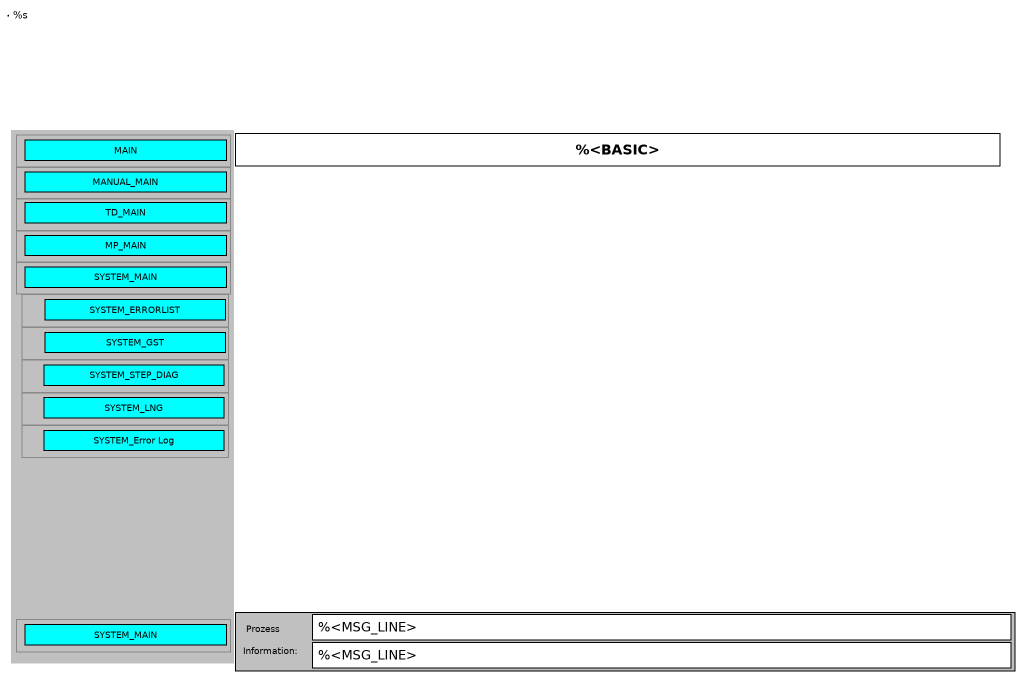
rectangle at (227,118)-(992,151): text "%<BASIC>"; shows 'Objekte ohne Grundstellung'
embedded screen at (3,115)-(226,648): M0003_System
rectangle at (227,597)-(1007,656): text "Prozess /  / Information:"
rectangle at (304,599)-(1003,625): text "%<MSG_LINE>"; shows ProcessMessage01
rectangle at (304,627)-(1003,653): text "%<MSG_LINE>"; shows ProcessMessage02
rectangle at (0,0)-(0,0): text "%s"; shows ListHomeNOK.HomeNOKArray[INDEX]
*)

(* Visualisation 04_System/SYSTEM_LNG
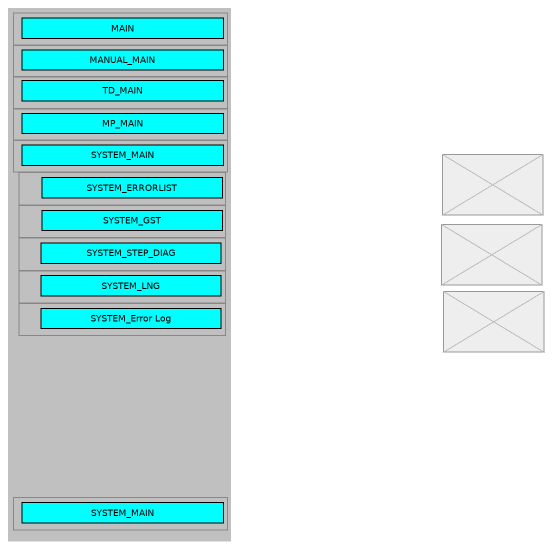
embedded screen at (3,115)-(226,648): M0003_System
bitmap at (437,261)-(538,322): bmp\de.bmp
bitmap at (436,331)-(537,392): bmp\en.bmp
bitmap at (438,398)-(539,459): bmp\cz.bmp
3 elements of other kinds (tables, trends, ...) not read
*)

(* Visualisation 04_System/SYSTEM_MAIN
